// TIA Portal V19 export
FUNCTION "A0302_Centratori_CALL" : Void   // FC97, LAD
// stored: SetENOAutomatically false
   VAR_TEMP
      Missing_Input : Bool;
      Missing_Output : Bool;
   END_VAR
BEGIN

REGION Network 1 (SCL): << TRASFERIMENTO stati CIn del blocco >>
   // SOSTITUIRE SYS BYPASS CON INGRESSI DIGITALI
   // TRASFERIMENTO COMANDI CIn MANAGER
   "A0302_Centratori".CIn.Manager := "A0302_Manager".COut.Rulliera.Centratori;
   //
   "A0302_Centratori".CIn.SemiAut_Pb := "A0302_Manager".DataIn.SemiAut_Pb;


   REGION TRASFERIMENTO STATI SENSORI RULLIERA 

       "A0302_Centratori".CIn.Rulliera.Coda.Sens.FTC_Rall := "A0302_Rulliera".IEC_FTC_CodaRall.FTC_On;
       "A0302_Centratori".CIn.Rulliera.Coda.Sens.FTC_Prox_Ing := "A0302_Rulliera".IEC_FTC_CodaProxIng.FTC_On;
       "A0302_Centratori".CIn.Rulliera.Centro.Sens.FTC_Centrale := "A0302_Rulliera".IEC_FTC_Centro.FTC_On;

   END_REGION ;

   REGION TRASFERIMENTO STATI CARRO PAREGGIATORE DI CODA

       "A0302_Centratori".CIn.CarroPareggCoda.Ax := "A0302_PareggiatoreCoda".COut.Ax;
       "A0302_Centratori".CIn.CarroPareggCoda.Bloccaggio := "A0302_PareggiatoreCoda".COut.Bloccaggio;
       "A0302_Centratori".CIn.CarroPareggCoda.BattutaVerticale := "A0302_PareggiatoreCoda".COut.BattutaVerticale;
       "A0302_Centratori".CIn.CarroPareggCoda.PareggiatoreLong := "A0302_PareggiatoreCoda".COut.PareggiatoreLong;
       "A0302_Centratori".CIn.CarroPareggCoda.Sens.FTC_Ingombro_In := "A0302_PareggiatoreCoda".IEC_FTC_Input.FTC_On;
       "A0302_Centratori".CIn.CarroPareggCoda.Sens.FTC_Ingombro_Out := "A0302_PareggiatoreCoda".IEC_FTC_Output.FTC_On;
       "A0302_Centratori".CIn.CarroPareggCoda.Sens.PresenzaMat := "A0302_PareggiatoreCoda".IEC_FTC_PresentMat.FTC_On;

   END_REGION ;

   REGION TRASFERIMENTO STATI CARRO PAREGGIATORE DI TESTA

       "A0302_Centratori".CIn.CarroPareggTesta.Ax := "A0302_PareggiatoreTesta".COut.Ax;
       "A0302_Centratori".CIn.CarroPareggTesta.Bloccaggio := "A0302_PareggiatoreTesta".COut.Bloccaggio;
       "A0302_Centratori".CIn.CarroPareggTesta.Centraggio := "A0302_PareggiatoreTesta".COut.Centraggio;
       "A0302_Centratori".CIn.CarroPareggTesta.Sollevatore := "A0302_PareggiatoreTesta".COut.Sollevatore;
       "A0302_Centratori".CIn.CarroPareggTesta.Sens.FTC1_Rall := "A0302_PareggiatoreTesta".IEC_FTC_Rall.FTC_On;
       "A0302_Centratori".CIn.CarroPareggTesta.Sens.FTC2_Prox_Ls := "A0302_PareggiatoreTesta".IEC_FTC_ProxLs.FTC_On;
       "A0302_Centratori".CIn.CarroPareggTesta.Sens.PresenzaMat := "A0302_PareggiatoreTesta".IEC_FTC_PresentMat.FTC_On;

   END_REGION ;

   // TRASFERIMENTO STATO DELLE ZONE INGRESSO E USCITA DELLA STAZIONE
   "A0302_Centratori".CIn.BTrk.ZoneA0302Entry_Empty := "A0302_Manager".Sts.BTrk.ZoneA0302Entry_Empty;
   "A0302_Centratori".CIn.BTrk.ZoneA0302Exit_Empty := "A0302_Manager".Sts.BTrk.ZoneA0302Exit_Empty;
END_REGION

REGION Network 2: <<< DATA IN >>>
END_REGION

REGION Network 3 (SCL): DATA In - Pulsanti OP
   // Pulsanti OP lavoro
   // 
   "A0302_Centratori".DataIn.OP.Rest := "A03_HMI".MB3.Button.A0302.Centratori.OP.Rest;
   "A0302_Centratori".DataIn.OP.Work := "A03_HMI".MB3.Button.A0302.Centratori.OP.Work;
END_REGION

REGION Network 4: DataIn - Centraggio 1
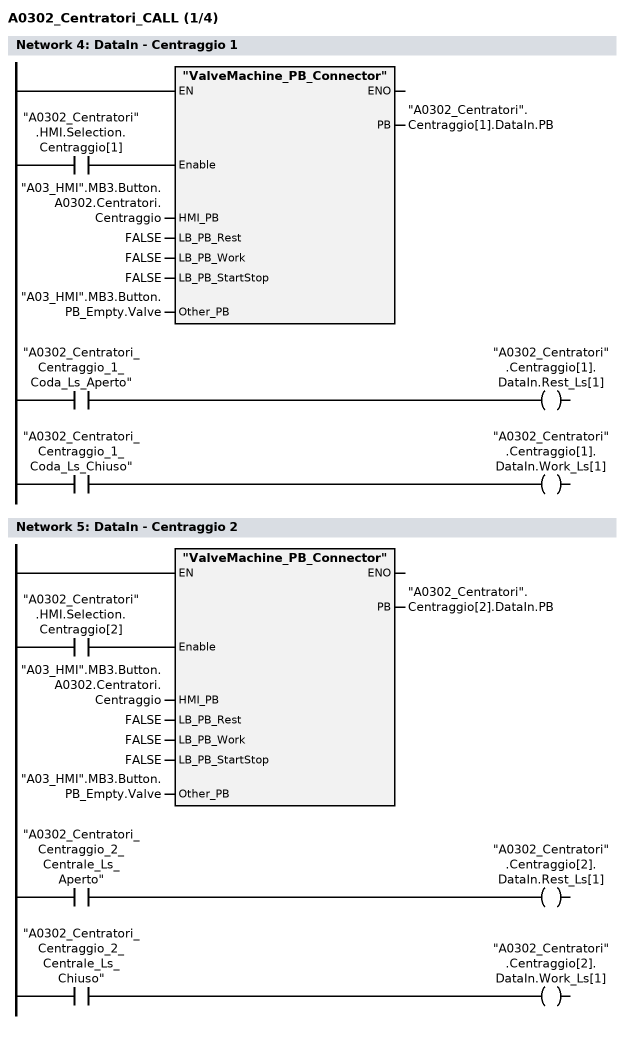
   RUNG wire#powerrail
      "ValveMachine_PB_Connector"(Enable := wire#w1, HMI_PB := "A03_HMI".MB3.Button.A0302.Centratori.Centraggio, LB_PB_Rest := FALSE, LB_PB_Work := FALSE, LB_PB_StartStop := FALSE, Other_PB := "A03_HMI".MB3.Button.PB_Empty.Valve, PB => "A0302_Centratori".Centraggio[1].DataIn.PB)
   END_RUNG
   RUNG wire#powerrail
      Contact( "A0302_Centratori".HMI.Selection.Centraggio[1] )
   END_RUNG wire#w1
   RUNG wire#powerrail
      Contact( "A0302_Centratori_Centraggio_1_Coda_Ls_Aperto" )
      Coil( "A0302_Centratori".Centraggio[1].DataIn.Rest_Ls[1] )
   END_RUNG
   RUNG wire#powerrail
      Contact( "A0302_Centratori_Centraggio_1_Coda_Ls_Chiuso" )
      Coil( "A0302_Centratori".Centraggio[1].DataIn.Work_Ls[1] )
   END_RUNG
   // the same network as SCL:
   "ValveMachine_PB_Connector"(Enable := "A0302_Centratori".HMI.Selection.Centraggio[1],
                           HMI_PB := "A03_HMI".MB3.Button.A0302.Centratori.Centraggio,
                           LB_PB_Rest := FALSE,
                           LB_PB_Work := FALSE,
                           LB_PB_StartStop := FALSE,
                           Other_PB := "A03_HMI".MB3.Button.PB_Empty.Valve,
                           PB => "A0302_Centratori".Centraggio[1].DataIn.PB);
   "A0302_Centratori".Centraggio[1].DataIn.Rest_Ls[1] := "A0302_Centratori_Centraggio_1_Coda_Ls_Aperto";
   "A0302_Centratori".Centraggio[1].DataIn.Work_Ls[1] := "A0302_Centratori_Centraggio_1_Coda_Ls_Chiuso";
END_REGION

REGION Network 5: DataIn - Centraggio 2
   RUNG wire#powerrail
      "ValveMachine_PB_Connector"(Enable := wire#w1, HMI_PB := "A03_HMI".MB3.Button.A0302.Centratori.Centraggio, LB_PB_Rest := FALSE, LB_PB_Work := FALSE, LB_PB_StartStop := FALSE, Other_PB := "A03_HMI".MB3.Button.PB_Empty.Valve, PB => "A0302_Centratori".Centraggio[2].DataIn.PB)
   END_RUNG
   RUNG wire#powerrail
      Contact( "A0302_Centratori".HMI.Selection.Centraggio[2] )
   END_RUNG wire#w1
   RUNG wire#powerrail
      Contact( "A0302_Centratori_Centraggio_2_Centrale_Ls_Aperto" )
      Coil( "A0302_Centratori".Centraggio[2].DataIn.Rest_Ls[1] )
   END_RUNG
   RUNG wire#powerrail
      Contact( "A0302_Centratori_Centraggio_2_Centrale_Ls_Chiuso" )
      Coil( "A0302_Centratori".Centraggio[2].DataIn.Work_Ls[1] )
   END_RUNG
   // the same network as SCL:
   "ValveMachine_PB_Connector"(Enable := "A0302_Centratori".HMI.Selection.Centraggio[2],
                           HMI_PB := "A03_HMI".MB3.Button.A0302.Centratori.Centraggio,
                           LB_PB_Rest := FALSE,
                           LB_PB_Work := FALSE,
                           LB_PB_StartStop := FALSE,
                           Other_PB := "A03_HMI".MB3.Button.PB_Empty.Valve,
                           PB => "A0302_Centratori".Centraggio[2].DataIn.PB);
   "A0302_Centratori".Centraggio[2].DataIn.Rest_Ls[1] := "A0302_Centratori_Centraggio_2_Centrale_Ls_Aperto";
   "A0302_Centratori".Centraggio[2].DataIn.Work_Ls[1] := "A0302_Centratori_Centraggio_2_Centrale_Ls_Chiuso";
END_REGION

REGION Network 6: DataIn - Centraggio 3
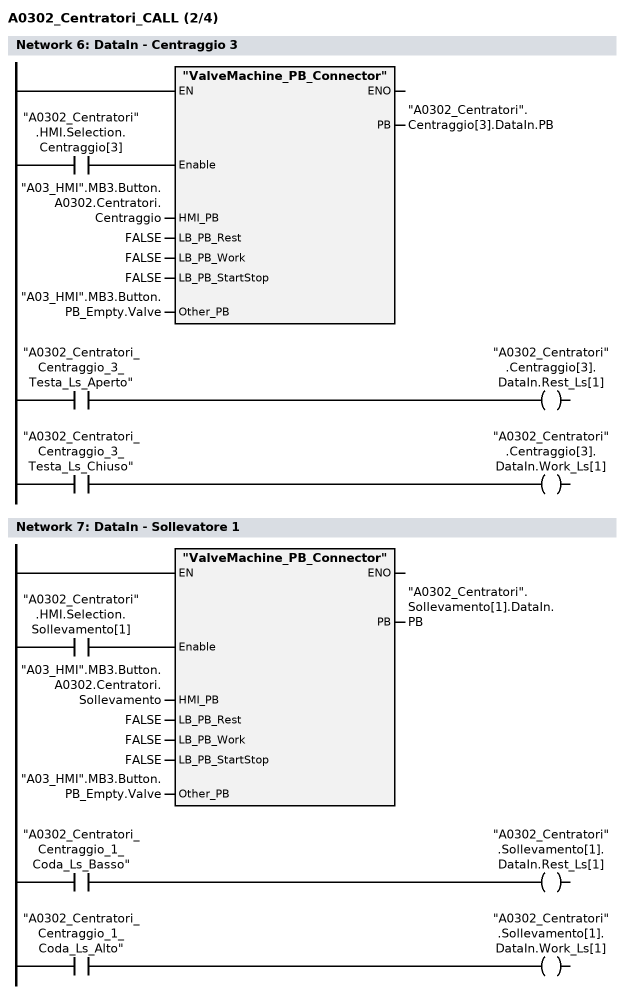
   RUNG wire#powerrail
      "ValveMachine_PB_Connector"(Enable := wire#w1, HMI_PB := "A03_HMI".MB3.Button.A0302.Centratori.Centraggio, LB_PB_Rest := FALSE, LB_PB_Work := FALSE, LB_PB_StartStop := FALSE, Other_PB := "A03_HMI".MB3.Button.PB_Empty.Valve, PB => "A0302_Centratori".Centraggio[3].DataIn.PB)
   END_RUNG
   RUNG wire#powerrail
      Contact( "A0302_Centratori".HMI.Selection.Centraggio[3] )
   END_RUNG wire#w1
   RUNG wire#powerrail
      Contact( "A0302_Centratori_Centraggio_3_Testa_Ls_Aperto" )
      Coil( "A0302_Centratori".Centraggio[3].DataIn.Rest_Ls[1] )
   END_RUNG
   RUNG wire#powerrail
      Contact( "A0302_Centratori_Centraggio_3_Testa_Ls_Chiuso" )
      Coil( "A0302_Centratori".Centraggio[3].DataIn.Work_Ls[1] )
   END_RUNG
   // the same network as SCL:
   "ValveMachine_PB_Connector"(Enable := "A0302_Centratori".HMI.Selection.Centraggio[3],
                           HMI_PB := "A03_HMI".MB3.Button.A0302.Centratori.Centraggio,
                           LB_PB_Rest := FALSE,
                           LB_PB_Work := FALSE,
                           LB_PB_StartStop := FALSE,
                           Other_PB := "A03_HMI".MB3.Button.PB_Empty.Valve,
                           PB => "A0302_Centratori".Centraggio[3].DataIn.PB);
   "A0302_Centratori".Centraggio[3].DataIn.Rest_Ls[1] := "A0302_Centratori_Centraggio_3_Testa_Ls_Aperto";
   "A0302_Centratori".Centraggio[3].DataIn.Work_Ls[1] := "A0302_Centratori_Centraggio_3_Testa_Ls_Chiuso";
END_REGION

REGION Network 7: DataIn - Sollevatore 1
   RUNG wire#powerrail
      "ValveMachine_PB_Connector"(Enable := wire#w1, HMI_PB := "A03_HMI".MB3.Button.A0302.Centratori.Sollevamento, LB_PB_Rest := FALSE, LB_PB_Work := FALSE, LB_PB_StartStop := FALSE, Other_PB := "A03_HMI".MB3.Button.PB_Empty.Valve, PB => "A0302_Centratori".Sollevamento[1].DataIn.PB)
   END_RUNG
   RUNG wire#powerrail
      Contact( "A0302_Centratori".HMI.Selection.Sollevamento[1] )
   END_RUNG wire#w1
   RUNG wire#powerrail
      Contact( "A0302_Centratori_Centraggio_1_Coda_Ls_Basso" )
      Coil( "A0302_Centratori".Sollevamento[1].DataIn.Rest_Ls[1] )
   END_RUNG
   RUNG wire#powerrail
      Contact( "A0302_Centratori_Centraggio_1_Coda_Ls_Alto" )
      Coil( "A0302_Centratori".Sollevamento[1].DataIn.Work_Ls[1] )
   END_RUNG
   // the same network as SCL:
   "ValveMachine_PB_Connector"(Enable := "A0302_Centratori".HMI.Selection.Sollevamento[1],
                           HMI_PB := "A03_HMI".MB3.Button.A0302.Centratori.Sollevamento,
                           LB_PB_Rest := FALSE,
                           LB_PB_Work := FALSE,
                           LB_PB_StartStop := FALSE,
                           Other_PB := "A03_HMI".MB3.Button.PB_Empty.Valve,
                           PB => "A0302_Centratori".Sollevamento[1].DataIn.PB);
   "A0302_Centratori".Sollevamento[1].DataIn.Rest_Ls[1] := "A0302_Centratori_Centraggio_1_Coda_Ls_Basso";
   "A0302_Centratori".Sollevamento[1].DataIn.Work_Ls[1] := "A0302_Centratori_Centraggio_1_Coda_Ls_Alto";
END_REGION

REGION Network 8: DataIn - Sollevatore 2
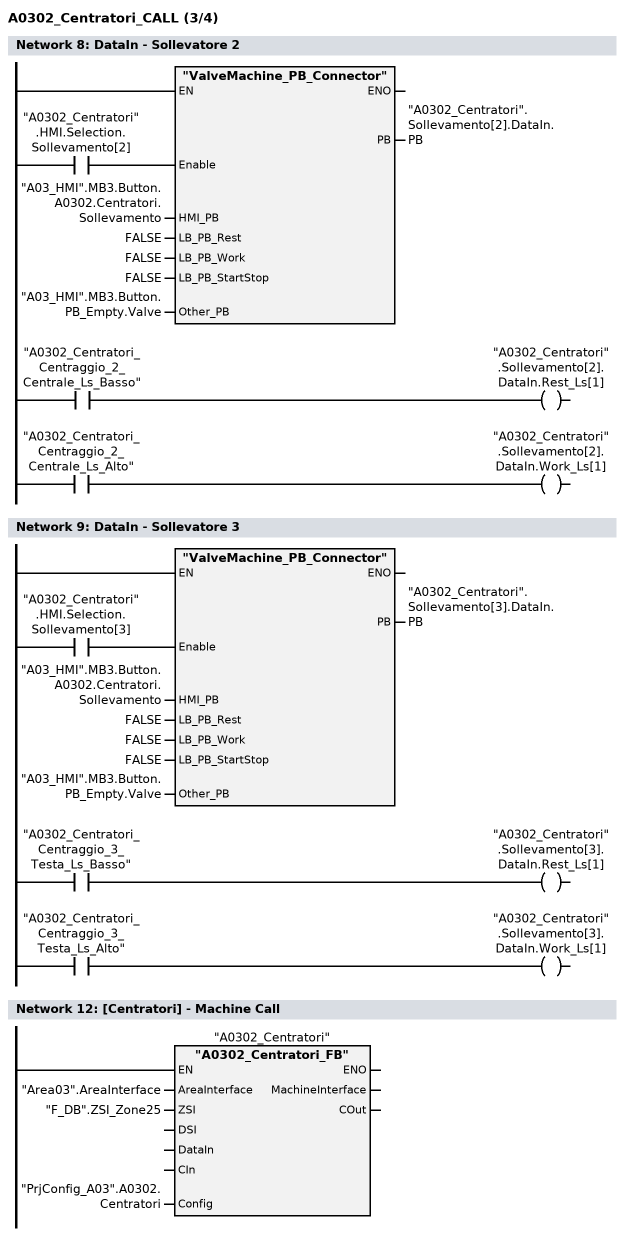
   RUNG wire#powerrail
      "ValveMachine_PB_Connector"(Enable := wire#w1, HMI_PB := "A03_HMI".MB3.Button.A0302.Centratori.Sollevamento, LB_PB_Rest := FALSE, LB_PB_Work := FALSE, LB_PB_StartStop := FALSE, Other_PB := "A03_HMI".MB3.Button.PB_Empty.Valve, PB => "A0302_Centratori".Sollevamento[2].DataIn.PB)
   END_RUNG
   RUNG wire#powerrail
      Contact( "A0302_Centratori".HMI.Selection.Sollevamento[2] )
   END_RUNG wire#w1
   RUNG wire#powerrail
      Contact( "A0302_Centratori_Centraggio_2_Centrale_Ls_Basso" )
      Coil( "A0302_Centratori".Sollevamento[2].DataIn.Rest_Ls[1] )
   END_RUNG
   RUNG wire#powerrail
      Contact( "A0302_Centratori_Centraggio_2_Centrale_Ls_Alto" )
      Coil( "A0302_Centratori".Sollevamento[2].DataIn.Work_Ls[1] )
   END_RUNG
   // the same network as SCL:
   "ValveMachine_PB_Connector"(Enable := "A0302_Centratori".HMI.Selection.Sollevamento[2],
                           HMI_PB := "A03_HMI".MB3.Button.A0302.Centratori.Sollevamento,
                           LB_PB_Rest := FALSE,
                           LB_PB_Work := FALSE,
                           LB_PB_StartStop := FALSE,
                           Other_PB := "A03_HMI".MB3.Button.PB_Empty.Valve,
                           PB => "A0302_Centratori".Sollevamento[2].DataIn.PB);
   "A0302_Centratori".Sollevamento[2].DataIn.Rest_Ls[1] := "A0302_Centratori_Centraggio_2_Centrale_Ls_Basso";
   "A0302_Centratori".Sollevamento[2].DataIn.Work_Ls[1] := "A0302_Centratori_Centraggio_2_Centrale_Ls_Alto";
END_REGION

REGION Network 9: DataIn - Sollevatore 3
   RUNG wire#powerrail
      "ValveMachine_PB_Connector"(Enable := wire#w1, HMI_PB := "A03_HMI".MB3.Button.A0302.Centratori.Sollevamento, LB_PB_Rest := FALSE, LB_PB_Work := FALSE, LB_PB_StartStop := FALSE, Other_PB := "A03_HMI".MB3.Button.PB_Empty.Valve, PB => "A0302_Centratori".Sollevamento[3].DataIn.PB)
   END_RUNG
   RUNG wire#powerrail
      Contact( "A0302_Centratori".HMI.Selection.Sollevamento[3] )
   END_RUNG wire#w1
   RUNG wire#powerrail
      Contact( "A0302_Centratori_Centraggio_3_Testa_Ls_Basso" )
      Coil( "A0302_Centratori".Sollevamento[3].DataIn.Rest_Ls[1] )
   END_RUNG
   RUNG wire#powerrail
      Contact( "A0302_Centratori_Centraggio_3_Testa_Ls_Alto" )
      Coil( "A0302_Centratori".Sollevamento[3].DataIn.Work_Ls[1] )
   END_RUNG
   // the same network as SCL:
   "ValveMachine_PB_Connector"(Enable := "A0302_Centratori".HMI.Selection.Sollevamento[3],
                           HMI_PB := "A03_HMI".MB3.Button.A0302.Centratori.Sollevamento,
                           LB_PB_Rest := FALSE,
                           LB_PB_Work := FALSE,
                           LB_PB_StartStop := FALSE,
                           Other_PB := "A03_HMI".MB3.Button.PB_Empty.Valve,
                           PB => "A0302_Centratori".Sollevamento[3].DataIn.PB);
   "A0302_Centratori".Sollevamento[3].DataIn.Rest_Ls[1] := "A0302_Centratori_Centraggio_3_Testa_Ls_Basso";
   "A0302_Centratori".Sollevamento[3].DataIn.Work_Ls[1] := "A0302_Centratori_Centraggio_3_Testa_Ls_Alto";
END_REGION

REGION Network 11 (SCL): DSI
   // Di solito facciamo struct DSI con dentro Centratori

   "A0302_Centratori".DSI := "F_DB".DSI_V_Air_A0302_A0303;
END_REGION

REGION Network 12: [Centratori] - Machine Call
   RUNG wire#powerrail
      "A0302_Centratori"(AreaInterface := "Area03".AreaInterface, ZSI := "F_DB".ZSI_Zone25, DSI :=, DataIn :=, CIn :=, Config := "PrjConfig_A03".A0302.Centratori, MachineInterface =>, COut =>)
   END_RUNG
   // the same network as SCL:
   "A0302_Centratori"(AreaInterface := "Area03".AreaInterface,   // "A0302_Centratori_FB"
                      ZSI := "F_DB".ZSI_Zone25,
                      Config := "PrjConfig_A03".A0302.Centratori);
END_REGION

REGION Network 14: <<< DATA OUT >>>
END_REGION

REGION Network 15: DataOut - Centraggio 1
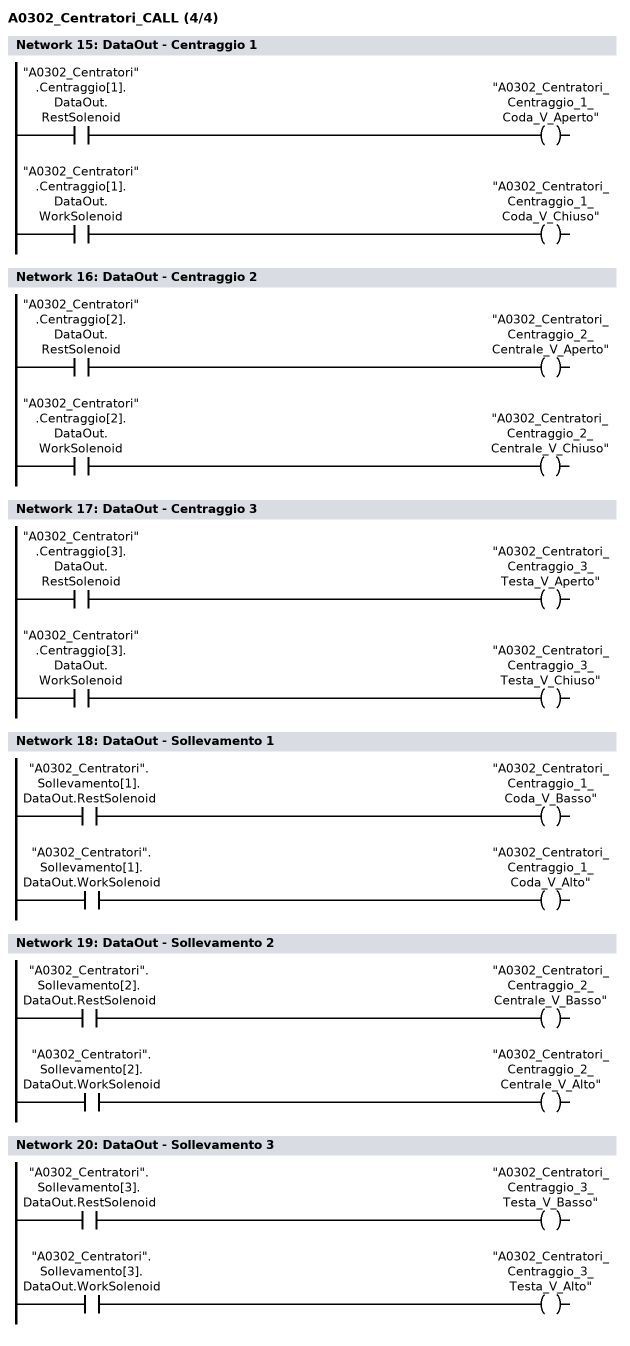
   RUNG wire#powerrail
      Contact( "A0302_Centratori".Centraggio[1].DataOut.RestSolenoid )
      Coil( "A0302_Centratori_Centraggio_1_Coda_V_Aperto" )
   END_RUNG
   RUNG wire#powerrail
      Contact( "A0302_Centratori".Centraggio[1].DataOut.WorkSolenoid )
      Coil( "A0302_Centratori_Centraggio_1_Coda_V_Chiuso" )
   END_RUNG
   // the same network as SCL:
   "A0302_Centratori_Centraggio_1_Coda_V_Aperto" := "A0302_Centratori".Centraggio[1].DataOut.RestSolenoid;
   "A0302_Centratori_Centraggio_1_Coda_V_Chiuso" := "A0302_Centratori".Centraggio[1].DataOut.WorkSolenoid;
END_REGION

REGION Network 16: DataOut - Centraggio 2
   RUNG wire#powerrail
      Contact( "A0302_Centratori".Centraggio[2].DataOut.RestSolenoid )
      Coil( "A0302_Centratori_Centraggio_2_Centrale_V_Aperto" )
   END_RUNG
   RUNG wire#powerrail
      Contact( "A0302_Centratori".Centraggio[2].DataOut.WorkSolenoid )
      Coil( "A0302_Centratori_Centraggio_2_Centrale_V_Chiuso" )
   END_RUNG
   // the same network as SCL:
   "A0302_Centratori_Centraggio_2_Centrale_V_Aperto" := "A0302_Centratori".Centraggio[2].DataOut.RestSolenoid;
   "A0302_Centratori_Centraggio_2_Centrale_V_Chiuso" := "A0302_Centratori".Centraggio[2].DataOut.WorkSolenoid;
END_REGION

REGION Network 17: DataOut - Centraggio 3
   RUNG wire#powerrail
      Contact( "A0302_Centratori".Centraggio[3].DataOut.RestSolenoid )
      Coil( "A0302_Centratori_Centraggio_3_Testa_V_Aperto" )
   END_RUNG
   RUNG wire#powerrail
      Contact( "A0302_Centratori".Centraggio[3].DataOut.WorkSolenoid )
      Coil( "A0302_Centratori_Centraggio_3_Testa_V_Chiuso" )
   END_RUNG
   // the same network as SCL:
   "A0302_Centratori_Centraggio_3_Testa_V_Aperto" := "A0302_Centratori".Centraggio[3].DataOut.RestSolenoid;
   "A0302_Centratori_Centraggio_3_Testa_V_Chiuso" := "A0302_Centratori".Centraggio[3].DataOut.WorkSolenoid;
END_REGION

REGION Network 18: DataOut - Sollevamento 1
   RUNG wire#powerrail
      Contact( "A0302_Centratori".Sollevamento[1].DataOut.RestSolenoid )
      Coil( "A0302_Centratori_Centraggio_1_Coda_V_Basso" )
   END_RUNG
   RUNG wire#powerrail
      Contact( "A0302_Centratori".Sollevamento[1].DataOut.WorkSolenoid )
      Coil( "A0302_Centratori_Centraggio_1_Coda_V_Alto" )
   END_RUNG
   // the same network as SCL:
   "A0302_Centratori_Centraggio_1_Coda_V_Basso" := "A0302_Centratori".Sollevamento[1].DataOut.RestSolenoid;
   "A0302_Centratori_Centraggio_1_Coda_V_Alto" := "A0302_Centratori".Sollevamento[1].DataOut.WorkSolenoid;
END_REGION

REGION Network 19: DataOut - Sollevamento 2
   RUNG wire#powerrail
      Contact( "A0302_Centratori".Sollevamento[2].DataOut.RestSolenoid )
      Coil( "A0302_Centratori_Centraggio_2_Centrale_V_Basso" )
   END_RUNG
   RUNG wire#powerrail
      Contact( "A0302_Centratori".Sollevamento[2].DataOut.WorkSolenoid )
      Coil( "A0302_Centratori_Centraggio_2_Centrale_V_Alto" )
   END_RUNG
   // the same network as SCL:
   "A0302_Centratori_Centraggio_2_Centrale_V_Basso" := "A0302_Centratori".Sollevamento[2].DataOut.RestSolenoid;
   "A0302_Centratori_Centraggio_2_Centrale_V_Alto" := "A0302_Centratori".Sollevamento[2].DataOut.WorkSolenoid;
END_REGION

REGION Network 20: DataOut - Sollevamento 3
   RUNG wire#powerrail
      Contact( "A0302_Centratori".Sollevamento[3].DataOut.RestSolenoid )
      Coil( "A0302_Centratori_Centraggio_3_Testa_V_Basso" )
   END_RUNG
   RUNG wire#powerrail
      Contact( "A0302_Centratori".Sollevamento[3].DataOut.WorkSolenoid )
      Coil( "A0302_Centratori_Centraggio_3_Testa_V_Alto" )
   END_RUNG
   // the same network as SCL:
   "A0302_Centratori_Centraggio_3_Testa_V_Basso" := "A0302_Centratori".Sollevamento[3].DataOut.RestSolenoid;
   "A0302_Centratori_Centraggio_3_Testa_V_Alto" := "A0302_Centratori".Sollevamento[3].DataOut.WorkSolenoid;
END_REGION
END_FUNCTION
